FUNCTION_BLOCK FB_Pump
VAR_INPUT
	command : BOOL ;
	feedback : BOOL ;
	auto_man : BOOL ;
	time_feedback : INT ;
END_VAR
VAR_OUTPUT
	valve: BOOL;	
END_VAR
VAR
	fbTimer: TON;
	fail : BOOL ;
END_VAR

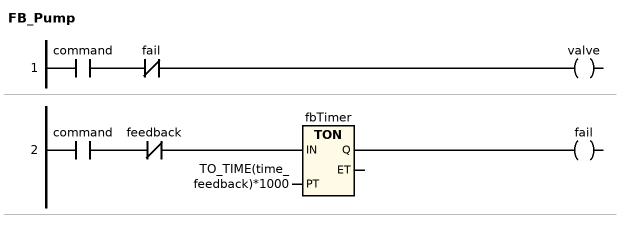
// NETWORK 1
valve := command AND NOT fail;

// NETWORK 2
fbTimer(IN := command AND NOT feedback, PT := TO_TIME(time_feedback)*1000); // TON
fail := fbTimer.Q;

END_FUNCTION_BLOCK

(* stored: Version 1.1.0.1, ProductVersion 3.1.4024.12
   POU FB_Pump: Id {b54b1369-fe0b-4219-9838-feacbf60322b}, SpecialFunc None *)
